(* PLC project v0.6.04_CycleSemiAuto.project, CODESYS CODESYS V3.5 SP19 Patch 1 *)
(* stored: creationDateTime 2026-08-11T14:02:33.687414, modificationDateTime 2026-08-11T14:02:33.687414 *)

(* ═══════════════════════════════════════════════════════════════ 🚦 ST_WinchState — États, mesures et diagnostics HMI pour un Treuil M1/M2 ─────────────────────────────────────────────────────────────── 🎨 Destiné aux retours d'informations et bargraphes HMI. ═══════════════════════════════════════════════════════════════ *)
TYPE ST_WinchState : STRUCT
  Position_M : REAL;  (* 🚦 États & Mesures (Lecture seule) 📊 Position actuelle du câble (mètres) *)
  MeasuredSpeed_Mps : REAL;  (* 📏 Vitesse linéaire mesurée du câble (m/s), valeur absolue *)
  SpeedDelta_Mps : REAL;  (* 🔍 Variation de vitesse entre deux scans (m/s) *)
  SpeedVariationDetected : BOOL;  (* 🔍 Seuil de variation dépassé sur le scan courant *)
  SpeedVariationConfirmed : BOOL;  (* 🛡️ Variation confirmée pendant la durée paramétrée *)
  SpeedStable : BOOL;  (* 🟢 Vitesse stable pendant la durée paramétrée *)
  SpeedMonitorError : BOOL;  (* 🔴 Défaut mémorisé du moniteur vitesse *)
  SpeedMonitorErrorId : WORD;  (* ❌ Bitfield du moniteur vitesse *)
  EstimatedLoadPct : REAL;  (* 📊 Estimation empirique, non certifiée *)
  LoadEstimateConfigured : BOOL;  (* 🟢 Table charge validée pour lecture *)
  SpeedGuardLimited : BOOL;  (* 🛡️ Palier limité par vitesse réelle *)
  SpeedRef_Pct : REAL;  (* 📈 Consigne de vitesse finale après rampe (%) *)
  StepNumber : INT;  (* 🔢 Palier de vitesse actif (0..5) *)
  FBState : E_State;  (* 🤖 État de l'automate interne (FB_Winch) *)
  Ready : BOOL;  (* 🟢 Treuil prêt à fonctionner *)
  Busy : BOOL;  (* ⚙️ Mouvement en cours *)
  Done : BOOL;  (* ✅ Action terminée *)
  Error : BOOL;  (* 🔴 Treuil en défaut *)
  ErrorId : WORD;  (* ❌ Code bitfield du défaut treuil *)
  RelayFwd : BOOL;  (* 🔌 Sorties Physiques / Indicateurs LEDs 🛗 Relais Montée activé *)
  RelayRev : BOOL;  (* 🛗 Relais Descente activé *)
  Contactor1 : BOOL;  (* 🔌 Contacteur vitesse palier 1 *)
  Contactor2 : BOOL;  (* 🔌 Contacteur vitesse palier 2 *)
  Contactor3 : BOOL;  (* 🔌 Contacteur vitesse palier 3 *)
  Contactor4 : BOOL;  (* 🔌 Contacteur vitesse palier 4 *)
  BrakeCmd : BOOL;  (* 🔓 Commande frein (TRUE = desserré / libre) *)
  FinalInterlockState : E_WinchFinalInterlockState;  (* 🛡️ État final _LD lecture seule *)
  FinalInterlockReason : E_WinchFinalInterlockReason;  (* 🛡️ Cause finale mémorisée *)
  FinalInterlockError : BOOL;  (* 🛡️ Défaut final mémorisé *)
  FinalInterlockErrorId : WORD;  (* 🛡️ Bitfield final *)
  FinalRestartInhibit : BOOL;  (* 🔒 Reset + neutre + nouvelle demande obligatoires *)
  BrakeCommandOpenConfirmed : BOOL;  (* 🔌 Contacteur/bobine desserrage confirmé, pas frein mécanique *)
  FinalAuthorizedStep : INT;  (* 🪜 Palier réellement autorisé *)
  FinalBrakeTimeoutElapsed : TIME;  (* ⏱️ Écoulé watchdog 500ms *)
  FinalRestartDelayElapsed : TIME;  (* ⏱️ Écoulé verrou redémarrage 900ms *)
  FinalStepDelayElapsed : TIME;  (* ⏱️ Écoulé entre paliers 1s250 *)
  Encoder : ST_EncoderHMI;  (* 🛡️ Sécurités & Diagnostics 🧲 Données d'échange et diagnostic du codeur — porte aussi les 9 champs Homing* (déplacés 2026-08, voir ST_EncoderHMI) *)
  ContactorsCheck : ST_ContactorCheck;  (* 🔍 Diagnostics de cohérence contacteurs réutilisés 🔌 Coherence contacteurs sens+vitesse *)
  BrakeContactorCheck : ST_ContactorCheck;  (* 🔌 Coherence retour frein *)
  InhibitActive : BOOL;  (* 🆕 miroir lecture seule — inhibition arbitrée *)
  BottomLimitActiveM : REAL;  (* 🐢 2026-08-07 : ralentissement sur bordure — diagnostic zone/limite active 📏 Limite basse active (m) — câble physique OU légale, la plus restrictive *)
  InTopSlowdownZone : BOOL;  (* 🐢 Palier plafonné à 1 : approche limite haute *)
  InBottomSlowdownZone : BOOL;  (* 🐢 Palier plafonné à 1 : approche limite basse (câble ou légale) *)
  CommandedDirection : INT;  (* 🩺 2026-08-07 : diagnostic retour terrain — délai ressenti à la remontée 🩺 Sens interne mémorisé FB_Winch (-1/0/+1) *)
  DirectionChangeDelayElapsed : TIME;  (* 🩺 Écoulé de l'interlock changement/reprise de sens *)
  DirectionChangePending : BOOL;  (* 🩺 TRUE tant que CommandedDirection n'a pas rejoint Direction *)
END_STRUCT;
END_TYPE

(* values of E_State: DISABLED: Enable faux, neutralisé; INIT: Démarrage / vérifs; READY: Prêt, attend ordre; BUSY: Action en cours; DONE: Action terminée; STOPPING: Décél rampe avant arrêt (StartStop=FALSE ou SafeStop=TRUE) *)

{attribute 'qualified_only'}
{attribute 'strict'}
TYPE E_State : (DISABLED := 0, INIT := 1, READY := 2, BUSY := 3, DONE := 4, STOPPING := 5);
END_TYPE

{attribute 'qualified_only'}
{attribute 'strict'}
TYPE E_WinchFinalInterlockReason : (NONE := 0, BRAKE_COMMAND_NOT_CONFIRMED := 1, RESTART_INHIBITED := 2);
END_TYPE

{attribute 'qualified_only'}
{attribute 'strict'}
TYPE E_WinchFinalInterlockState : (DISABLED := 0, READY := 1, WAIT_BRAKE_COMMAND_CONFIRMATION := 2, WAIT_STEP_DELAY := 3, WAIT_RESTART_DELAY := 4, FAULT := 5);
END_TYPE

(* ═══════════════════════════════════════════════════════════════ 🔌 ST_ContactorCheck — Double vérification commande/retour contacteur ─────────────────────────────────────────────────────────────── 📄 Doc métier : DOC/AF/AF_Partie-02_Architecture_Programme_v3.1.md §3, DOC/AF/AF_Partie-03_Contrats_Composants_v2.1.md §2 Utilisé par FB_Brake (frein) et FB_Winch (contacteurs de sens) pour détecter un collage / une absence de fermeture d'un contacteur de puissance, au-delà d'un délai de cohérence (FeedbackTimeout du FB appelant). ═══════════════════════════════════════════════════════════════ *)
TYPE ST_ContactorCheck : STRUCT
  Command : BOOL;  (* Ordre envoyé au contacteur (TRUE = fermé/actif) *)
  Feedback : BOOL;  (* Retour d'état câblé (TRUE = effectivement fermé) *)
  StuckClosed : BOOL;  (* Diag : commande OFF mais retour ON depuis trop longtemps → PowerCutOff *)
  StuckOpen : BOOL;  (* Diag : commande ON mais retour OFF depuis trop longtemps *)
END_STRUCT;
END_TYPE

(* ═══════════════════════════════════════════════════════════════ 🧲 ST_EncoderHMI — Données d'échange IHM pour les codeurs absolus ─────────────────────────────────────────────────────────────── 🎨 Destiné à l'affichage des informations et diagnostics des codeurs. ═══════════════════════════════════════════════════════════════ *)
TYPE ST_EncoderHMI : STRUCT
  RawPos : UDINT;  (* 📊 Position brute lue sur le bus *)
  Alarms : UINT;  (* ⚠️ Code d'alarme brut du codeur *)
  Warnings : UINT;  (* 🟧 Code d'avertissement brut du codeur *)
  SlaveOperational : BOOL;  (* 📡 Esclave EtherCAT opérationnel *)
  PresetTriggerCmd : WORD;  (* 🎯 Commande de preset active *)
  PresetValueOut : UDINT;  (* 📐 Valeur de preset envoyée au codeur *)
  Error : BOOL;  (* 🔴 Codeur en défaut (liaison EtherCAT ou preset) *)
  ErrorId : WORD;  (* ❌ Code défaut codeur *)
  Homed : BOOL;  (* 🎯 Homing — déplacés depuis ST_WinchState racine (2026-08, réorganisation ST_WinchHMI/Homing) 🎯 Prise d'origine (Homing) validée *)
  HomingBusy : BOOL;  (* ⏳ Référencement en cours *)
  HomingDone : BOOL;  (* ✅ Pulse de référencement réussi *)
  HomingError : BOOL;  (* 🔴 Défaut de référencement *)
  HomingErrorId : WORD;  (* ❌ Bitfield défaut homing *)
  HomingState : E_State;  (* 🤖 État FB_Encoder_Homing *)
  HomingStateAtError : E_State;  (* 🧭 État lors du défaut *)
  HomingSuspect : BOOL;  (* ⚠️ Référence à confirmer *)
  HomingRefRaw : UDINT;  (* 📐 Référence brute appliquée *)
END_STRUCT;
END_TYPE
